(* PLC project MotionTest1, Higen MCL 1 *)
(* stored: creationDateTime 2012-01-06T15:20:13, modificationDateTime 2026-03-05T12:13:59 *)

PROGRAM main
  VAR
    clock : ULINT;
    Done : BOOL;
    Axis : AXIS_REF;
    moveA : MC_MoveAbsolute;
    switch : MC_Power;
    readpos : MC_ReadActualPosition;
    Pn : LREAL;
    Vn : LREAL;
    setpos : MC_SetPosition;
    readspeed : MC_ReadParameter;
    moveB : MC_Stop;
    movead : MC_MoveAdditive;
    my_sim : MC_Sim;
  END_VAR

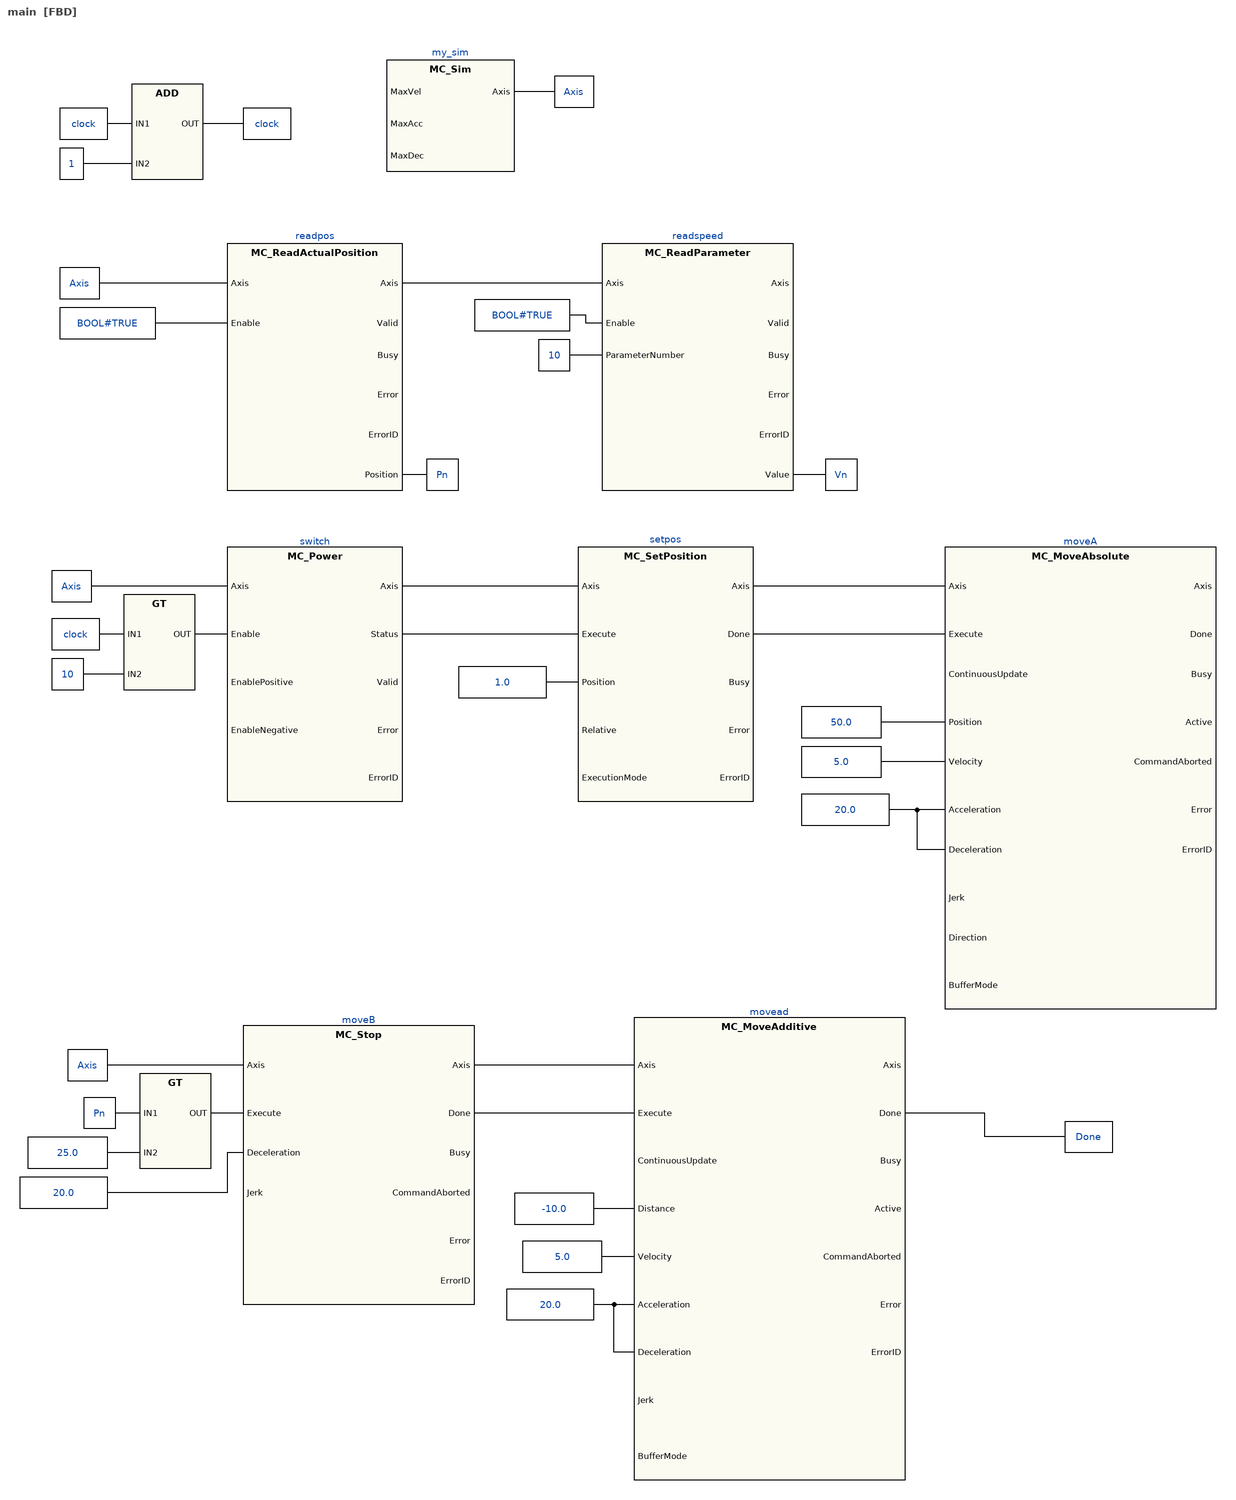
(* FBD diagram, written out as Structured Text *)
clock := clock + 1;
readpos(Axis := Axis, Enable := BOOL#TRUE);
Pn := readpos.Position;
readspeed(Axis := readpos.Axis, Enable := BOOL#TRUE, ParameterNumber := 10);
Vn := readspeed.Value;
moveB(Axis := Axis, Execute := Pn > 25.0, Deceleration := 20.0);
movead(Axis := moveB.Axis, Execute := moveB.Done, Distance := -10.0, Velocity := 5.0, Acceleration := 20.0, Deceleration := 20.0);
Done := movead.Done;
my_sim();
Axis := my_sim.Axis;
switch(Axis := Axis, Enable := clock > 10);
setpos(Axis := switch.Axis, Execute := switch.Status, Position := 1.0);
moveA(Axis := setpos.Axis, Execute := setpos.Done, Position := 50.0, Velocity := 5.0, Acceleration := 20.0, Deceleration := 20.0);
END_PROGRAM

CONFIGURATION conf
  RESOURCE res ON PLC
    TASK milisecond(INTERVAL := T#1ms, PRIORITY := 0);
    PROGRAM maininstance WITH milisecond : main;
  END_RESOURCE
END_CONFIGURATION
